FUNCTION CAN_Receive : BOOL
VAR_INPUT
END_VAR
VAR
	// CAN-BUS
	arrCobId : ARRAY [0..45]OF UINT;
	arrCobIdTmp : ARRAY [0..45]OF UINT;
	MessageReceived: ARRAY [0..9] OF CANQUEUE;
	test_number_1 : REAL;
	test_number_2 : REAL;
	test : CANQUEUE;
	MsgId : UINT;
	// Indexing vars
	i: UINT;
	j : UINT;

	z: UINT;
	n: INT;
	z_old: UINT;
END_VAR

(* Receiving, CAN-BUS *)
IF Outputs.TxQueue.RxCounter <> Inputs.RxQueue.RxCounter THEN
	FOR i := 0 TO (Inputs.RxQueue.NoOfRxMessages-1) DO
		MessageReceived[i] := Inputs.RxQueue.RxMessages[i];
	END_FOR
	Outputs.TxQueue.RxCounter := Outputs.TxQueue.RxCounter+1;
END_IF

(*
IF (Inputs.NoOfRxMessages = 0) THEN
	RETURN;
END_IF
*)


(*Parsing*)
FOR z:=0 TO (Inputs.RxQueue.NoOfRxMessages) DO
	 (*Logging last 45 received CobId's*)
	IF z<>z_old AND n<45 THEN
		arrCobId[n]:=MessageReceived[z].cobId;
		IF n>=44 THEN n:=0;arrCobIdTmp:=arrCobId; ELSE n:=n+1; END_IF
		z_old:=z;
	END_IF
	
	//Removes the last five bits in number and shifts five places
	MsgId := SHR(MessageReceived[z].cobId AND 16#FFE0, 5);

	(*Case structure to catch specific CobId and parse data from it*)
	CASE  MsgId OF		
			
		40: (* Engine Oil Pressure *)
			test := MessageReceived[z];
			
		//ELSE // DEBUG
		//	J1939_UNKNOWN_COBID	:=MessageReceived[z];
		//	J1939_createVisString(rxData:=ADR(MessageReceived[z].rxData) , strRxData=>strJ1939_UNKNOWN_COBID );
			// DISPLAY UNKNOW MESSAGES
	//		ADSLOGSTR(msgCtrlMask:=ADSLOG_MSGTYPE_HINT , msgFmtStr:= 'J1939 uknown CobId: ' , strArg:=strJ1939_UNKNOWN_COBID );
	
		200:
			ByteArrayToReal(MessageReceived[z],0, output => test_number_1);
			ByteArrayToReal(MessageReceived[z],4, output => test_number_2);
		
		201:
			ByteArrayToDINT(MessageReceived[z], 0, output => Process.PumpOpen);
			
		202:
			ByteArrayToDINT(MessageReceived[z], 0, output => Process.HoistingEnable);
			ByteArrayToReal(MessageReceived[z], 4, output => Process.HoistingDemandValue);
			
		203:
			ByteArrayToDINT(MessageReceived[z], 0, output => Process.PumpEnable);
			ByteArrayToReal(MessageReceived[z], 4, output => Process.PumpPID);
			
		206:
			ByteArrayToReal(MessageReceived[z], 0, output => Process.InputTopDriveRPMSetPoint);
			ByteArrayToReal(MessageReceived[z], 4, output => Process.InputTopDriveTorqueSetPoint);
			
		208:
			ByteArrayToDINT(MessageReceived[z], 0, output => Process.TopDriveEnable);
	END_CASE
END_FOR

END_FUNCTION

(* stored: Version 1.1.0.1, ProductVersion 3.1.4024.9
   POU CAN_Receive: Id {aeb3c2e1-15ab-4af4-9092-f5a8cf50f535}, SpecialFunc None *)
